TYPE ST_NciChannel_Ref :
STRUCT
  NcToPlc AT %I*: NcToPlc_NciChannel_Ref;   //  Externer Datentyp!
  PlcToNc AT %Q*: PlcToNc_NciChannel_Ref;   //  Externer Datentyp!
END_STRUCT
END_TYPE

(* stored: Version 1.1.0.1, ProductVersion 3.1.4024.12
   DUT ST_NciChannel_Ref: Id {18b59b54-3056-08a9-0a40-0372544b635f} *)
